TYPE ST_SlaveState :
STRUCT
    (* slave state *)
    eEcState 		: E_EcCommState;
    nReserved		: UINT;
    bError			: BOOL;
    bInvalidVPRS	: BOOL;
    nReserved2		: UINT;

    (* link state *)
    bNoCommToSlave	: BOOL;
    bLinkError		: BOOL;
    bMissingLink	: BOOL;
    bUnexpectedLink	: BOOL;
    bPortA			: BOOL;
    bPortB			: BOOL;
    bPortC			: BOOL;
    bPortD			: BOOL;
END_STRUCT
END_TYPE

(* stored: Version 1.1.0.1
   DUT ST_SlaveState: Id {95acdbd0-e32f-4597-b051-9455dffeea2c} *)
